DECL E6POS XP172={X 1340.88623,Y -402.247284,Z 1672.75110,A 0.846814,B -44.5353661,C -108.428535,S 2,T 34,E1 -15.0944824,E2 195.002243,E3 195.004120,E4 0.0,E5 0.0,E6 0.0}
DECL FDAT FP172={TOOL_NO 1,BASE_NO 0,IPO_FRAME #BASE,POINT2[] " ",TQ_STATE FALSE}
DECL PDAT PPDAT127={VEL 100.000,ACC 100.000,APO_DIST 100.000,APO_MODE #CDIS,GEAR_JERK 50.0000,EXAX_IGN 3}
DECL E6POS XP173={X 1319.30261,Y -675.391785,Z 1607.84973,A 5.64195442,B -41.0563393,C -122.908539,S 0,T 34,E1 -15.0944824,E2 195.002243,E3 195.004120,E4 0.0,E5 0.0,E6 0.0}
DECL FDAT FP173={TOOL_NO 1,BASE_NO 0,IPO_FRAME #BASE,POINT2[] " ",TQ_STATE FALSE}
DECL PDAT PPDAT128={VEL 100.000,ACC 100.000,APO_DIST 100.000,APO_MODE #CDIS,GEAR_JERK 50.0000,EXAX_IGN 3}
DECL E6POS XP174={X 1340.88623,Y -402.247284,Z 1672.75110,A 0.846814,B -44.5353661,C -108.428535,S 2,T 34,E1 -15.0944824,E2 195.002243,E3 195.004120,E4 0.0,E5 0.0,E6 0.0}
DECL FDAT FP174={TOOL_NO 1,BASE_NO 0,IPO_FRAME #BASE,POINT2[] " ",TQ_STATE FALSE}
DECL PDAT PPDAT129={VEL 100.000,ACC 100.000,APO_DIST 100.000,APO_MODE #CDIS,GEAR_JERK 50.0000,EXAX_IGN 3}
DECL ATBg_Start_T AS_WDAT92={JobModeId -187662529,ParamSetId 687014726,StartTime 0.0,PreFlowTime 0.100000,Channel1 30.0000,Channel2 1.00000,Channel3 0.0,Channel4 0.0,Channel5 0.0,Channel6 0.0,Channel7 0.0,Channel8 0.0,PurgeTime 0.0}
DECL ATBg_Weld_T AW_WDAT92={JobModeId -187662529,ParamSetId -430485013,Velocity 0.00830000,Channel1 30.0000,Channel2 1.00000,Channel3 0.0,Channel4 0.0,Channel5 0.0,Channel6 0.0,Channel7 0.0,Channel8 0.0}
DECL WTCg_WeaveDefinition_T WV_WDAT92={Pattern #None,Length 4.00000,Amplitude 2.00000,Angle 0.0}
DECL FDAT FP175={TOOL_NO 1,BASE_NO 0,IPO_FRAME #BASE,POINT2[] " ",TQ_STATE FALSE}
DECL PDAT PPDAT130={ACC 100.000,APO_DIST 100.000,APO_MODE #CPTP,GEAR_JERK 50.0000}
DECL E6POS XP175={X 1473.60986,Y -91.8296127,Z 1579.61023,A -3.94931197,B -41.4006348,C -87.8952255,S 2,T 42,E1 -15.0945082,E2 195.002151,E3 195.004089,E4 0.0,E5 0.0,E6 0.0}
DECL ATBg_Crater_T AC_WDAT93={JobModeId -187662529,ParamSetId -1375177600,CraterTime 0.100000,PostflowTime 0.100000,Channel1 30.0000,Channel2 1.00000,Channel3 0.0,Channel4 0.0,Channel5 0.0,Channel6 0.0,Channel7 0.0,Channel8 0.0,BurnBackTime 0.0}
DECL FDAT FP176={TOOL_NO 1,BASE_NO 0,IPO_FRAME #BASE,POINT2[] " ",TQ_STATE FALSE}
DECL LDAT LCPDAT49={ACC 100.000,APO_DIST 100.000,APO_FAC 50.0000,AXIS_VEL 100.000,AXIS_ACC 100.000,ORI_TYP #VAR,CIRC_TYP #BASE,JERK_FAC 50.0000,GEAR_JERK 50.0000,EXAX_IGN 0}
DECL E6POS XP176={X 1473.60986,Y -91.8296127,Z 1579.61023,A -3.94931197,B -41.4006348,C -87.8952255,S 2,T 42,E1 -15.0945082,E2 195.002151,E3 195.004089,E4 0.0,E5 0.0,E6 0.0}
DECL ATBg_Start_T AS_WDAT94={JobModeId -187662529,ParamSetId 687014726,StartTime 0.0,PreFlowTime 0.100000,Channel1 30.0000,Channel2 1.00000,Channel3 0.0,Channel4 0.0,Channel5 0.0,Channel6 0.0,Channel7 0.0,Channel8 0.0,PurgeTime 0.0}
DECL ATBg_Weld_T AW_WDAT94={JobModeId -187662529,ParamSetId -430485013,Velocity 0.00830000,Channel1 30.0000,Channel2 1.00000,Channel3 0.0,Channel4 0.0,Channel5 0.0,Channel6 0.0,Channel7 0.0,Channel8 0.0}
DECL WTCg_WeaveDefinition_T WV_WDAT94={Pattern #None,Length 4.00000,Amplitude 2.00000,Angle 0.0}
DECL FDAT FP177={TOOL_NO 1,BASE_NO 0,IPO_FRAME #BASE,POINT2[] " ",TQ_STATE FALSE}
DECL PDAT PPDAT131={ACC 100.000,APO_DIST 100.000,APO_MODE #CPTP,GEAR_JERK 50.0000}
DECL E6POS XP177={X 1467.48669,Y 163.778198,Z 1580.61816,A 7.33355141,B -41.5764198,C -91.4063950,S 2,T 43,E1 -15.0945082,E2 195.002151,E3 195.004089,E4 0.0,E5 0.0,E6 0.0}
DECL ATBg_Crater_T AC_WDAT95={JobModeId -187662529,ParamSetId -1375177600,CraterTime 0.100000,PostflowTime 0.100000,Channel1 30.0000,Channel2 1.00000,Channel3 0.0,Channel4 0.0,Channel5 0.0,Channel6 0.0,Channel7 0.0,Channel8 0.0,BurnBackTime 0.0}
DECL FDAT FP178={TOOL_NO 1,BASE_NO 0,IPO_FRAME #BASE,POINT2[] " ",TQ_STATE FALSE}
DECL LDAT LCPDAT50={ACC 100.000,APO_DIST 100.000,APO_FAC 50.0000,AXIS_VEL 100.000,AXIS_ACC 100.000,ORI_TYP #VAR,CIRC_TYP #BASE,JERK_FAC 50.0000,GEAR_JERK 50.0000,EXAX_IGN 0}
DECL E6POS XP178={X 1467.48669,Y 163.778198,Z 1580.61816,A 7.33355141,B -41.5764198,C -91.4063950,S 2,T 43,E1 -15.0945082,E2 195.002151,E3 195.004089,E4 0.0,E5 0.0,E6 0.0}
DECL E6POS XP179={X 1301.48328,Y 149.157791,Z 1778.32690,A 7.88870478,B -52.9349670,C -92.1586151,S 2,T 43,E1 -15.0945082,E2 195.002151,E3 195.004089,E4 0.0,E5 0.0,E6 0.0}
DECL FDAT FP179={TOOL_NO 1,BASE_NO 0,IPO_FRAME #BASE,POINT2[] " ",TQ_STATE FALSE}
DECL PDAT PPDAT132={VEL 100.000,ACC 100.000,APO_DIST 100.000,APO_MODE #CDIS,GEAR_JERK 50.0000,EXAX_IGN 3}
DECL ATBg_Start_T AS_WDAT96={JobModeId -187662529,ParamSetId 687014726,StartTime 0.0,PreFlowTime 0.100000,Channel1 30.0000,Channel2 1.00000,Channel3 0.0,Channel4 0.0,Channel5 0.0,Channel6 0.0,Channel7 0.0,Channel8 0.0,PurgeTime 0.0}
DECL ATBg_Weld_T AW_WDAT96={JobModeId -187662529,ParamSetId -430485013,Velocity 0.00830000,Channel1 30.0000,Channel2 1.00000,Channel3 0.0,Channel4 0.0,Channel5 0.0,Channel6 0.0,Channel7 0.0,Channel8 0.0}
DECL WTCg_WeaveDefinition_T WV_WDAT96={Pattern #None,Length 4.00000,Amplitude 2.00000,Angle 0.0}
DECL FDAT FP180={TOOL_NO 1,BASE_NO 0,IPO_FRAME #BASE,POINT2[] " ",TQ_STATE FALSE}
DECL PDAT PPDAT133={ACC 100.000,APO_DIST 100.000,APO_MODE #CPTP,GEAR_JERK 50.0000}
DECL E6POS XP180={X 1406.94678,Y 538.867798,Z 1576.37537,A -1.21830094,B -38.4161911,C -71.3365860,S 2,T 43,E1 -15.0945082,E2 195.002151,E3 195.004089,E4 0.0,E5 0.0,E6 0.0}
DECL ATBg_Crater_T AC_WDAT97={JobModeId -187662529,ParamSetId -1375177600,CraterTime 0.100000,PostflowTime 0.100000,Channel1 30.0000,Channel2 1.00000,Channel3 0.0,Channel4 0.0,Channel5 0.0,Channel6 0.0,Channel7 0.0,Channel8 0.0,BurnBackTime 0.0}
DECL FDAT FP181={TOOL_NO 1,BASE_NO 0,IPO_FRAME #BASE,POINT2[] " ",TQ_STATE FALSE}
DECL LDAT LCPDAT51={ACC 100.000,APO_DIST 100.000,APO_FAC 50.0000,AXIS_VEL 100.000,AXIS_ACC 100.000,ORI_TYP #VAR,CIRC_TYP #BASE,JERK_FAC 50.0000,GEAR_JERK 50.0000,EXAX_IGN 0}
DECL E6POS XP181={X 1406.94678,Y 538.867798,Z 1576.37537,A -1.21830094,B -38.4161911,C -71.3365860,S 2,T 43,E1 -15.0945082,E2 195.002151,E3 195.004089,E4 0.0,E5 0.0,E6 0.0}
DECL E6POS XP182={X 1239.22363,Y 477.509247,Z 1777.01758,A -5.46240807,B -48.6917725,C -65.2049179,S 0,T 43,E1 -15.0945082,E2 195.002151,E3 195.004089,E4 0.0,E5 0.0,E6 0.0}
DECL FDAT FP182={TOOL_NO 1,BASE_NO 0,IPO_FRAME #BASE,POINT2[] " ",TQ_STATE FALSE}
DECL PDAT PPDAT134={VEL 100.000,ACC 100.000,APO_DIST 100.000,APO_MODE #CDIS,GEAR_JERK 50.0000,EXAX_IGN 3}
DECL E6POS XP183={X 1239.22363,Y 477.509247,Z 1777.01758,A -5.46240807,B -48.6917725,C -65.2049179,S 0,T 43,E1 -15.0945082,E2 195.002151,E3 195.004089,E4 0.0,E5 0.0,E6 0.0}
DECL FDAT FP183={TOOL_NO 1,BASE_NO 0,IPO_FRAME #BASE,POINT2[] " ",TQ_STATE FALSE}
DECL PDAT PPDAT135={VEL 100.000,ACC 100.000,APO_DIST 100.000,APO_MODE #CDIS,GEAR_JERK 50.0000,EXAX_IGN 3}
DECL E6POS XP184={X 1374.48206,Y 155.586990,Z 1703.80115,A 7.64417267,B -48.7668076,C -91.8435059,S 2,T 43,E1 -15.0945082,E2 195.002151,E3 195.004089,E4 0.0,E5 0.0,E6 0.0}
DECL FDAT FP184={TOOL_NO 1,BASE_NO 0,IPO_FRAME #BASE,POINT2[] " ",TQ_STATE FALSE}
DECL PDAT PPDAT136={VEL 100.000,ACC 100.000,APO_DIST 100.000,APO_MODE #CDIS,GEAR_JERK 50.0000,EXAX_IGN 3}
DECL E6POS XP185={X 1297.61536,Y -75.5030289,Z 1792.50964,A -3.57095265,B -54.1264305,C -88.4031143,S 2,T 42,E1 -15.0945082,E2 195.002151,E3 195.004089,E4 0.0,E5 0.0,E6 0.0}
DECL FDAT FP185={TOOL_NO 1,BASE_NO 0,IPO_FRAME #BASE,POINT2[] " ",TQ_STATE FALSE}
DECL PDAT PPDAT137={VEL 100.000,ACC 100.000,APO_DIST 100.000,APO_MODE #CDIS,GEAR_JERK 50.0000,EXAX_IGN 3}
ENDDAT
